FUNCTION_BLOCK ConveyorCTLMulti (* Basic Function Block Type *)
  (* Standard: 61499-2 *)
  (* Version 0.2, 2003-12-04, JHC, Rockwell Automation, Renamed for better indexing. *)
  (* Version 0.1, 2002-11-05, JHC, Rockwell Automation, Corrected missing ST element in Algorithm REQ. *)
  (* Version 0.0, 2000-05-30, JHC, Rockwell Automation *)
  (* Compiler header: package fb.rt.cs725; *)
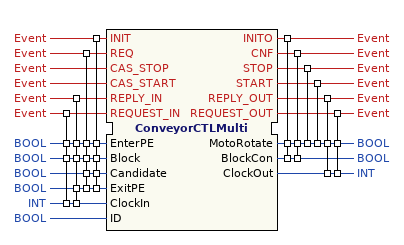
  EVENT_INPUT
    INIT WITH Block, Candidate, ExitPE, EnterPE; (* Initialization Request *)
    REQ WITH EnterPE, Block, Candidate, ExitPE; (* Normal Execution Request *)
    CAS_STOP;
    CAS_START;
    REPLY_IN WITH ExitPE, EnterPE, Block, ClockIn;
    REQUEST_IN WITH EnterPE, Block, ClockIn;
  END_EVENT
  EVENT_OUTPUT
    INITO WITH MotoRotate, BlockCon; (* Initialization Confirm *)
    CNF WITH MotoRotate, BlockCon; (* Execution Confirmation *)
    STOP WITH MotoRotate;
    START WITH MotoRotate;
    REPLY_OUT WITH MotoRotate, ClockOut;
    REQUEST_OUT WITH MotoRotate, ClockOut;
  END_EVENT
  VAR_INPUT
    EnterPE : BOOL; (* Input event qualifier *)
    Block : BOOL;
    Candidate : BOOL;
    ExitPE : BOOL;
    ClockIn : INT;
    ID : BOOL;
  END_VAR
  VAR_OUTPUT
    MotoRotate : BOOL; (* Output event qualifier *)
    BlockCon : BOOL;
    ClockOut : INT;
  END_VAR
  VAR
    lastPE : BOOL := 1;
    lastBlock : BOOL := 0;
    StoreEmit : BOOL := 0;
    CLOCK : INT;
    Priority : BOOL;
  END_VAR
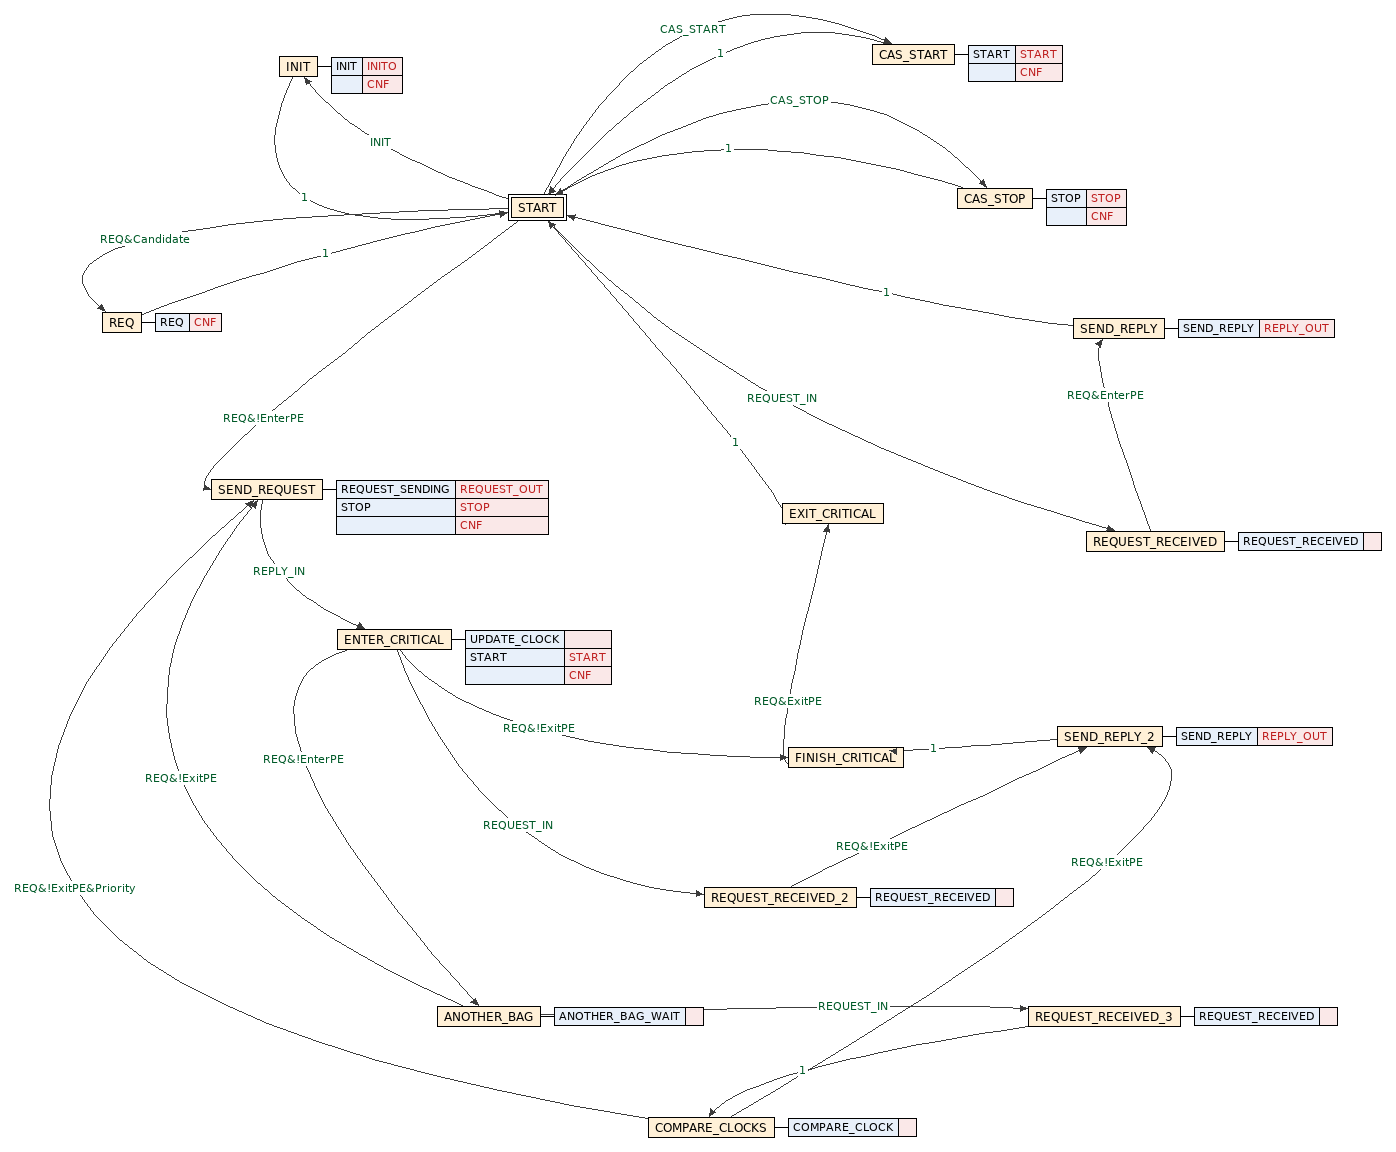
  EC_STATES
    START; (* Initial State *)
    INIT : INIT -> INITO, -> CNF; (* Initialization *)
    CAS_START : START -> START, -> CNF;
    CAS_STOP : STOP -> STOP, -> CNF;
    SEND_REQUEST : REQUEST_SENDING -> REQUEST_OUT, STOP -> STOP, -> CNF;
    ENTER_CRITICAL : UPDATE_CLOCK, START -> START, -> CNF;
    FINISH_CRITICAL;
    EXIT_CRITICAL;
    REQUEST_RECEIVED : REQUEST_RECEIVED;
    SEND_REPLY : SEND_REPLY -> REPLY_OUT;
    REQ : REQ -> CNF;
    REQUEST_RECEIVED_2 : REQUEST_RECEIVED;
    SEND_REPLY_2 : SEND_REPLY -> REPLY_OUT;
    ANOTHER_BAG : ANOTHER_BAG_WAIT;
    REQUEST_RECEIVED_3 : REQUEST_RECEIVED;
    COMPARE_CLOCKS : COMPARE_CLOCK;
  END_STATES
  EC_TRANSITIONS
    START TO INIT := INIT;
    INIT TO START := 1;
    START TO CAS_START := CAS_START;
    CAS_START TO START := 1;
    START TO CAS_STOP := CAS_STOP;
    CAS_STOP TO START := 1;
    START TO SEND_REQUEST := REQ&!EnterPE;
    SEND_REQUEST TO ENTER_CRITICAL := REPLY_IN;
    ENTER_CRITICAL TO FINISH_CRITICAL := REQ&!ExitPE;
    FINISH_CRITICAL TO EXIT_CRITICAL := REQ&ExitPE;
    EXIT_CRITICAL TO START := 1;
    START TO REQUEST_RECEIVED := REQUEST_IN;
    SEND_REPLY TO START := 1;
    REQUEST_RECEIVED TO SEND_REPLY := REQ&EnterPE;
    START TO REQ := REQ&Candidate;
    REQ TO START := 1;
    ENTER_CRITICAL TO REQUEST_RECEIVED_2 := REQUEST_IN;
    REQUEST_RECEIVED_2 TO SEND_REPLY_2 := REQ&!ExitPE;
    SEND_REPLY_2 TO FINISH_CRITICAL := 1;
    ENTER_CRITICAL TO ANOTHER_BAG := REQ&!EnterPE;
    ANOTHER_BAG TO SEND_REQUEST := REQ&!ExitPE;
    ANOTHER_BAG TO REQUEST_RECEIVED_3 := REQUEST_IN;
    REQUEST_RECEIVED_3 TO COMPARE_CLOCKS := 1;
    COMPARE_CLOCKS TO SEND_REQUEST := REQ&!ExitPE&Priority;
    COMPARE_CLOCKS TO SEND_REPLY_2 := REQ&!ExitPE;
  END_TRANSITIONS
  ALGORITHM INIT IN ST: (* Initialization algorithm *)
MotoRotate := TRUE;
Block := FALSE;
  END_ALGORITHM
  ALGORITHM REQ IN ST: (* Normally executed algorithm *)
IF Candidate THEN
IF lastPE !:= EnterPE THEN
IF NOT EnterPE THEN
BlockCon:= TRUE;
System.out.println("BlockCon = true");
ELSE
BlockCon:=FALSE;
System.out.println("BlockCon = false");
END_IF
lastPE := EnterPE;
END_IF
IF lastBlock !:= Block THEN
IF Block THEN
STOP.serviceEvent(this);
MotoRotate := FALSE;
System.out.println("Cas Stop");
ELSE
START.serviceEvent(this);
MotoRotate := TRUE;
System.out.println("Cas Start");
END_IF
lastBlock := Block;
END_IF
END_IF
  END_ALGORITHM
  ALGORITHM START IN ST:
MotoRotate:=TRUE;
  END_ALGORITHM
  ALGORITHM STOP IN ST:
MotoRotate := FALSE;
  END_ALGORITHM
  ALGORITHM REQUEST_SENDING IN Java:
System.out.println("Requesting for Multicast");
  END_ALGORITHM
  ALGORITHM ANOTHER_BAG_WAIT IN Java:
System.out.println("Another bag is wating for multicast");
  END_ALGORITHM
  ALGORITHM REQUEST_RECEIVED IN Java:
System.out.println("Multicast received a new request");
  END_ALGORITHM
  ALGORITHM SEND_REPLY IN Java:
System.out.println("Replied to Multicast request");
  END_ALGORITHM
  ALGORITHM DIFFERENT_REQUEST IN Java:
System.out.println("Request from another conveyer received");
  END_ALGORITHM
  ALGORITHM COMPARE_CLOCK IN Java:
System.out.println("Comparing clocks");
if(ClockIn.value>CLOCK.value){
Priority.value=true;
}
else {
Priority.value=false;
}
  END_ALGORITHM
  ALGORITHM UPDATE_CLOCK IN Java:
CLOCK.value++;
ClockOut.value = CLOCK.value;
System.out.printf("Clock value updated = %d%n",CLOCK.value);
  END_ALGORITHM
END_FUNCTION_BLOCK
